FUNCTION MA_Velocity_Slave : INT

VAR_INPUT
	//Enable: BOOL:=0;
	Speed: REAL:=0;
	Disturbance: REAL:=0;
END_VAR


VAR_IN_OUT
	Axis: Motion_Axis;
END_VAR

VAR
	i: INT:=0;
END_VAR

Axis.IN_Closed_Open_Loop:=1;
Axis.IN_Enable_Control:=1;

Axis.OL_IN_Analog:=0;
Axis.OL_IN_Slave_Enable:=0;
Axis.OL_Move_Type:=0;
Axis.OL_IN_Bump_Duration:= T#0MS;  //Timer for Bump Type of Move
Axis.OL_IN_Bump_Trigger:= 0;

Axis.CL_IN_Vel:=Speed;
Axis.CL_IN_Slave_Enable:=1;
Axis.CL_IN_Slave_Command:=Disturbance;
Axis.CL_IN_Vary_Vel:=0;
Axis.CL_IN_Load:=0;
Axis.CL_Move_Type:=1;

END_FUNCTION

(* stored: Version 1.1.0.1, ProductVersion 3.1.4020.12
   POU MA_Velocity_Slave: Id {78feb408-c3f6-44a1-aa5a-314c8fadcd58}, SpecialFunc None *)
